// TIA Portal V17 export
// export: Created 2023-02-25T14:39:32.5815196Z, ExportSetting WithDefaults, DisplayName Totally Integrated Automation Portal, DisplayVersion V17, DisplayName TIA Portal Openness, DisplayVersion V17, DisplayName TIA Portal Version Control Interface, DisplayVersion V17, DisplayName TIA Portal Test Suite Advanced, DisplayVersion V17, DisplayName STEP 7 Professional, DisplayVersion V17, DisplayName SIMATIC Energy Suite, DisplayVersion V17, DisplayName STEP 7 Safety, DisplayVersion V17, DisplayName WinCC Professional, DisplayVersion V17
DATA_BLOCK "HW_HardwareData"   // DB16
{ S7_Optimized_Access := 'TRUE' }
VERSION : 0.1
// stored: AutoNumber true, IsOnlyStoredInLoadMemory false, IsRetainMemResEnabled false, IsWriteProtectedInAS false, MemoryReserve 100
   VAR
      C1 : "stt_Motor";
      C2 { S7_SetPoint := 'True'} : "stt_Motor";
      C3 { S7_SetPoint := 'True'} : "stt_Motor";
      C4 { S7_SetPoint := 'True'} : "stt_Motor";
      W { S7_SetPoint := 'True'} : Bool;
      SendLeft : Bool;
      SendForward : Bool;
      SendRight : Bool;
   END_VAR
BEGIN
END_DATA_BLOCK
